PROGRAM B_Program
VAR
	i : UINT;
	x : LREAL;
	x_inc : LREAL := 0.0001;
END_VAR

FOR i := 0 TO 100 DO
	x := x + x_inc;
END_FOR

END_PROGRAM

(* stored: Version 1.1.0.1, ProductVersion 3.1.4025.12
   POU B_Program: Id {a7c33278-aeef-48eb-8fcf-05960a00375d}, SpecialFunc None *)
